// TIA Portal V20 export
DATA_BLOCK "Data_block_1"   // DB1
TITLE = Motor
{ S7_Optimized_Access := 'TRUE' }
// stored: MemoryReserve 100
   VAR
      Motor_on : Bool := false;
      Motor_overload : Bool;
      Target_position : Int := 50;
   END_VAR
BEGIN
END_DATA_BLOCK
